FUNCTION_BLOCK FB_Press
VAR_IN_OUT

AxisPressing :AXIS_REF;//扭矩轴
Press_SystemRUN  :ST_SystemRUN;//热、冷压系统
Clear_press    :BOOL;//压力清零信号
Permit_Press   :BOOL;//允许热、冷压信号
Press_Finish   :BOOL;//热、冷压完成信号

END_VAR
	
VAR_INPUT
	Step: UINT;
	AxisPress	 :INT;//扭矩轴名称
	AxisTensed	 :INT;//麦拉膜轴名称
	CylinderPress	:INT;//麦拉膜气缸名称
	Press_M          :INT;//电芯记忆名称
	Press_SV :REAL;//当前压力值
	Press_P  :REAL;//压力调节值P值
	Press_I  :REAL;//压力调节值I值
	Press_D  :REAL;//压力调节值D值
	AD_Press :INT;//压力模拟量
	Press_Factor :REAL;//扭矩系数
	Torque_Offset :REAL;//扭矩偏移量
	TorqueRamp    :REAL;//扭矩变化率 
	VelocityLimit :REAL;//扭矩速度限制
	Press_Time :INT;//保持压力时间

END_VAR

VAR_OUTPUT
	Press_PV :REAL;//当前压力值
	Torque_Act :REAL;//扭矩当前值
END_VAR

VAR
Press_H_Limit :REAL;//压力上限值
Press_L_Limit :REAL;//压力下限值
Press_max     :REAL;//压力最大值
Press_min     :REAL;//压力最小值
Press_PID_Out :REAL;//PID输出值	
FB_MC_TorqueControl_1: MC_TorqueControl;
FB_MC_MoveVelocity_1: MC_MoveVelocity;
Hot_Torque: INT;
FB_Unwinding_PID_1: Unwinding_PID;
Press_Time_Z:TIME;
Press_TON :TON;
FB_MC_Stop_1: MC_Stop;
END_VAR

Press_PV:=INT_TO_REAL(AD_Press)*4;
Press_max:=Press_SV+1000;
Press_min:=Press_SV-400;
Torque_Act:=Press_PV*Press_Factor+Torque_Offset;
FB_MC_TorqueControl_1.Torque:=REAL_TO_LREAL(Press_SV*Press_Factor);
FB_MC_TorqueControl_1.TorqueRamp:=REAL_TO_LREAL(TorqueRamp);
FB_MC_TorqueControl_1.VelocityLimitHigh:=REAL_TO_LREAL(VelocityLimit+5);
FB_MC_TorqueControl_1.VelocityLimitLow:=REAL_TO_LREAL(VelocityLimit);

FB_MC_MoveVelocity_1.Velocity:=-Press_PID_Out*REAL#0.5;
FB_MC_MoveVelocity_1.Acceleration:=FB_MC_MoveVelocity_1.Velocity*10;
FB_MC_MoveVelocity_1.Deceleration:=FB_MC_MoveVelocity_1.Velocity*10;
FB_MC_MoveVelocity_1.Jerk:=FB_MC_MoveVelocity_1.Velocity*100;
FB_MC_MoveVelocity_1.Velocity:=LIMIT(-LREAL#2,FB_MC_MoveVelocity_1.Velocity,LREAL#2);
Press_Time_Z:=INT_TO_TIME(Press_Time);

IF Press_SystemRUN.iMode=1 THEN
CASE Step OF
1://驱动电机回初始位	
IF  NOT arrAxisCtrl[AxisPress].Cmd.arrbRealPoint[1] AND NOT arrAxisCtrl[AxisPress].Status.Error AND arrAxisCtrl[AxisPress].Status.Homed 
	AND arrAxisCtrl[AxisPress].Status.Enabled AND arrAxisCtrl[AxisPress].Status.NoMoving THEN
	arrAxisCtrl[AxisPress].Cmd.iGoSetPos:=1;
END_IF 

IF arrAxisCtrl[AxisPress].Cmd.arrbRealPoint[1]	AND arrAxisCtrl[AxisPress].Status.NoMoving THEN
	Step:=5;
	Clear_press:=TRUE;//压力清零信号
END_IF

5://判断是否能热、冷压

IF Permit_Press AND NOT CellMemory[Press_M].ScanCode=2 THEN
	Step:=10;
	Clear_press:=FALSE;
END_IF


10://麦拉膜轴去张开位和麦拉膜气缸张紧
arrCyCtrl[CylinderPress].Cmd.bON:=TRUE;
IF  arrAxisCtrl[AxisPress].Cmd.arrbRealPoint[1]	AND
	NOT arrAxisCtrl[AxisTensed].Cmd.arrbRealPoint[2] AND NOT arrAxisCtrl[AxisTensed].Status.Error AND arrAxisCtrl[AxisTensed].Status.Homed 
	AND arrAxisCtrl[AxisTensed].Status.Enabled AND arrAxisCtrl[AxisTensed].Status.NoMoving THEN
	arrAxisCtrl[AxisTensed].Cmd.iGoSetPos:=2;	
END_IF
 IF arrAxisCtrl[AxisTensed].Cmd.arrbRealPoint[2] AND arrAxisCtrl[AxisTensed].Status.NoMoving AND arrCyCtrl[CylinderPress].Status.ONState 
	AND NOT arrCyCtrl[CylinderPress].Status.Error1 THEN
	step:=20;
END_IF

20://扭矩轴去电芯位

IF NOT arrAxisCtrl[AxisPress].Cmd.arrbRealPoint[2] AND NOT arrAxisCtrl[AxisPress].Status.Error AND arrAxisCtrl[AxisPress].Status.Homed 
	AND arrAxisCtrl[AxisPress].Status.Enabled AND arrAxisCtrl[AxisPress].Status.NoMoving THEN
	arrAxisCtrl[AxisPress].Cmd.iGoSetPos:=2;	
END_IF 

IF arrAxisCtrl[AxisPress].Cmd.arrbRealPoint[2]	AND Permit_Press AND arrAxisCtrl[AxisPress].Status.NoMoving THEN
	Step:=30;
END_IF

30://开始走扭矩
FB_MC_TorqueControl_1.Execute:=TRUE;
IF FB_MC_TorqueControl_1.InTorque AND Press_PV>Press_min AND Press_PV<Press_max THEN//扭矩达到范围值开始走PID
	Step:=40;
	FB_MC_TorqueControl_1.Execute:=FALSE;
END_IF

40://保压
FB_MC_MoveVelocity_1.Execute:=TRUE;//走PID
Press_TON.PT:=Press_Time_Z;
Press_TON.IN:=TRUE;
IF Press_TON.Q THEN//保压时间达到后
	Step:=50;
	Press_TON.IN:=FALSE;
	FB_MC_MoveVelocity_1.Execute:=FALSE;
END_IF
	
50://轴停止
FB_MC_Stop_1.Execute:=TRUE;
IF FB_MC_Stop_1.Done THEN
	Step:=60;
	FB_MC_Stop_1.Execute:=FALSE;
END_IF

60://扭矩轴回初始位
IF  NOT arrAxisCtrl[AxisPress].Cmd.arrbRealPoint[1] AND NOT arrAxisCtrl[AxisPress].Status.Error AND arrAxisCtrl[AxisPress].Status.Homed 
	AND arrAxisCtrl[AxisPress].Status.Enabled AND arrAxisCtrl[AxisPress].Status.NoMoving THEN
	arrAxisCtrl[AxisPress].Cmd.iGoSetPos:=1;	
END_IF 
IF arrAxisCtrl[AxisPress].Cmd.arrbRealPoint[1] AND arrAxisCtrl[AxisPress].Status.NoMoving THEN
	Permit_Press :=FALSE;//复位允许冷、热压信号
	Press_Finish:=TRUE;//冷热压完成信号可以下料
	Step:=70;
END_IF

70:
Step:=1;

END_CASE
END_IF

ACTION TorqueAndPID:
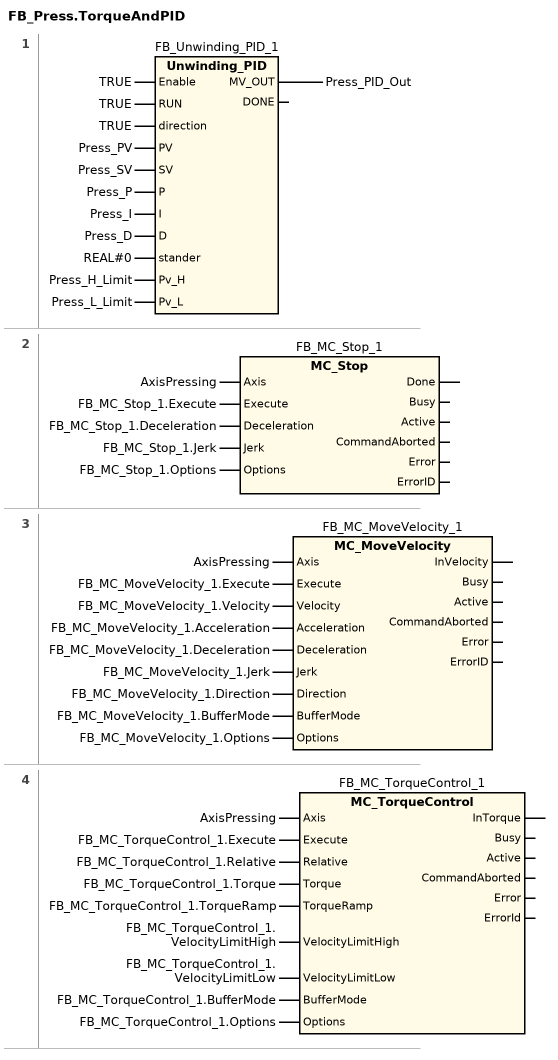
// NETWORK 1
FB_Unwinding_PID_1(
    Enable := TRUE,
    RUN := TRUE,
    direction := TRUE,
    PV := Press_PV,
    SV := Press_SV,
    P := Press_P,
    I := Press_I,
    D := Press_D,
    stander := REAL#0,
    Pv_H := Press_H_Limit,
    Pv_L := Press_L_Limit); // Unwinding_PID
Press_PID_Out := FB_Unwinding_PID_1.MV_OUT;

// NETWORK 2
FB_MC_Stop_1(
    Axis := AxisPressing,
    Execute := FB_MC_Stop_1.Execute,
    Deceleration := FB_MC_Stop_1.Deceleration,
    Jerk := FB_MC_Stop_1.Jerk,
    Options := FB_MC_Stop_1.Options); // MC_Stop

// NETWORK 3
FB_MC_MoveVelocity_1(
    Axis := AxisPressing,
    Execute := FB_MC_MoveVelocity_1.Execute,
    Velocity := FB_MC_MoveVelocity_1.Velocity,
    Acceleration := FB_MC_MoveVelocity_1.Acceleration,
    Deceleration := FB_MC_MoveVelocity_1.Deceleration,
    Jerk := FB_MC_MoveVelocity_1.Jerk,
    Direction := FB_MC_MoveVelocity_1.Direction,
    BufferMode := FB_MC_MoveVelocity_1.BufferMode,
    Options := FB_MC_MoveVelocity_1.Options); // MC_MoveVelocity

// NETWORK 4
FB_MC_TorqueControl_1(
    Axis := AxisPressing,
    Execute := FB_MC_TorqueControl_1.Execute,
    Relative := FB_MC_TorqueControl_1.Relative,
    Torque := FB_MC_TorqueControl_1.Torque,
    TorqueRamp := FB_MC_TorqueControl_1.TorqueRamp,
    VelocityLimitHigh := FB_MC_TorqueControl_1.VelocityLimitHigh,
    VelocityLimitLow := FB_MC_TorqueControl_1.VelocityLimitLow,
    BufferMode := FB_MC_TorqueControl_1.BufferMode,
    Options := FB_MC_TorqueControl_1.Options); // MC_TorqueControl
END_ACTION

END_FUNCTION_BLOCK

(* stored: Version 1.1.0.1, ProductVersion 3.1.4024.9
   POU FB_Press: Id {ad1766a7-453c-4ec2-94e7-f3d712c98b93}, SpecialFunc None
   Action TorqueAndPID: Id {9b270b8a-8c15-4584-a763-2385e5a6fcd3} *)
